FUNCTION_BLOCK FB_UvLedModule IMPLEMENTS I_DeviceBase
VAR_INPUT
  IbReady                  AT%I* : BOOL;
END_VAR

VAR_OUTPUT
  ObEnableHigh             AT%Q* : BOOL;
  ObLowIntenseMode         AT%Q* : BOOL;
  ObDisableLeft            AT%Q* : BOOL;
  ObDisableRight           AT%Q* : BOOL;
  OnIntensitySetpoint      AT%Q* : WORD;  (*Setpoint for intensity control  [digit]*)
END_VAR

VAR
  _bActivate                     : BOOL;
  _sName                         : STRING := '';
  _nColorRGB                     : UDINT;
  _sColorName                    : STRING := 'undef';    (*color name*)
END_VAR

VAR CONSTANT
  CnAnalogMinDigit               : DINT := 0;      (*Min value analog-output in digit*)
  CnAnalogMaxDigit               : DINT := 32767;  (*Max value analog-output in digit*)
  CnMinIntensitySetpoint         : DINT := 5;      (*Min setpoint for intensity control [%]*)
  CnMaxIntensitySetpoint         : DINT := 100;    (*Max setpoint for intensity control [%]*)
END_VAR

VAR PERSISTENT
  RbLowIntenseMode               : BOOL := FALSE;  (*Visu: set low intense mode*)
  RbDisableLeft                  : BOOL := FALSE;  (*Visu: disable left SLM*)
  RbDisableRight                 : BOOL := FALSE;  (*Visu: disable right SLM*)
  RnIntensitySetpoint            : DINT := 20;     (*Visu: setpoint for intensity control [%]*)
END_VAR

(*Set outputs*)
ObEnableHigh        := _bActivate;
ObLowIntenseMode    := RbLowIntenseMode;
ObDisableLeft       := RbDisableLeft;
ObDisableRight      := RbDisableRight;
OnIntensitySetpoint := DINT_TO_WORD(CnAnalogMaxDigit * RnIntensitySetpoint / 100);  (*Setpoint [digit]*)

METHOD Init : BOOL
VAR_INPUT
  nColorRGB    : UDINT;     (*color RGB*)
  sColorName   : STRING;    (*color name*)
END_VAR
_nColorRGB := nColorRGB;
_sColorName := sColorName;
END_METHOD

METHOD mDisable : BOOL
_bActivate := FALSE;
END_METHOD

METHOD mEnable : BOOL
_bActivate := TRUE;
END_METHOD

{attribute 'monitoring':='call'}
PROPERTY pActive : BOOL
GET
pActive := _bActivate;
END_GET
END_PROPERTY

PROPERTY pErrorCode : INT
GET
pErrorCode := 0;  // no error
END_GET
END_PROPERTY

END_FUNCTION_BLOCK

(* stored: Version 1.1.0.1, ProductVersion 3.1.4024.11
   POU FB_UvLedModule: Id {3f4eca81-28a1-427b-8cc1-b934d6bded93}, SpecialFunc None
   Folder I_DeviceBase: Id {8d640c35-7667-43b9-bfa3-25a0453f0d8d}
   Method Init: Id {4ec47f5d-f08c-48cb-9a2b-d64c9c7b11ba}
   Method mDisable: Id {69edd295-f260-4933-889c-986f73e3fd12}
   Method mEnable: Id {e7faa1d3-d717-40dd-97e1-4128d21d4838}
   Property pActive: Id {5a931f28-b826-4eb9-8a20-33a2db125118}
   Get Get: Id {254f1391-79b3-4938-91e5-575bba5fa1e4}
   Property pErrorCode: Id {1aefa6c7-005a-42f8-870b-575a1eb8da43}
   Get Get: Id {ad16c2ce-f00c-49bb-98f2-b73fd3b2d0cf} *)
